// Mitsubishi GX Works2 project: MPS 장비 제어 4   PLC: Q03UDV

PROGRAM MAIN
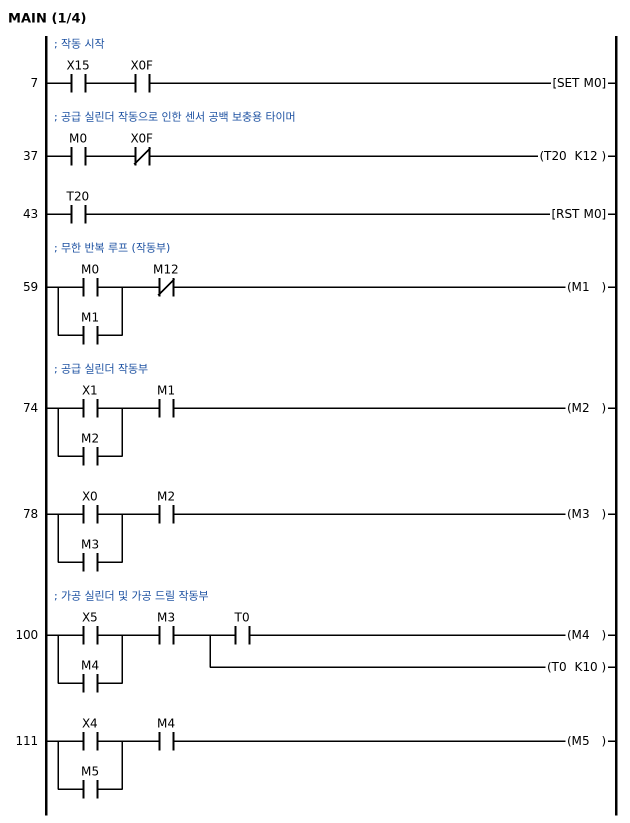
; 작동 시작
7     LD      X15
      AND     X0F
      SET     M0
; 공급 실린더 작동으로 인한 센서 공백 보충용 타이머
37    LD      M0
      ANI     X0F
      OUT     T20 K12
43    LD      T20
      RST     M0
; 무한 반복 루프 (작동부)
59    LD      M0
      OR      M1
      ANI     M12
      OUT     M1
; 공급 실린더 작동부
74    LD      X1
      OR      M2
      AND     M1
      OUT     M2
78    LD      X0
      OR      M3
      AND     M2
      OUT     M3
; 가공 실린더 및 가공 드릴 작동부
100   LD      X5
      OR      M4
      AND     M3
      MPS
      AND     T0
      OUT     M4
      MPP
      OUT     T0 K10
111   LD      X4
      OR      M5
      AND     M4
      OUT     M5
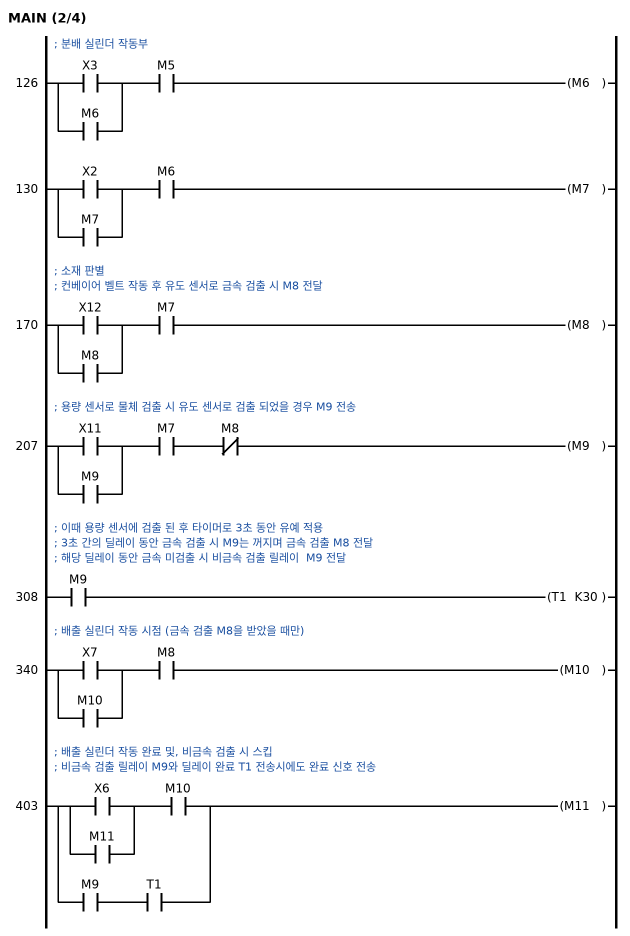
; 분배 실린더 작동부
126   LD      X3
      OR      M6
      AND     M5
      OUT     M6
130   LD      X2
      OR      M7
      AND     M6
      OUT     M7
; 소재 판별
; 컨베이어 벨트 작동 후 유도 센서로 금속 검출 시 M8 전달
170   LD      X12
      OR      M8
      AND     M7
      OUT     M8
; 용량 센서로 물체 검출 시 유도 센서로 검출 되었을 경우 M9 전송
207   LD      X11
      OR      M9
      AND     M7
      ANI     M8
      OUT     M9
; 이때 용량 센서에 검출 된 후 타이머로 3초 동안 유예 적용
; 3초 간의 딜레이 동안 금속 검출 시 M9는 꺼지며 금속 검출 M8 전달
; 해당 딜레이 동안 금속 미검출 시 비금속 검출 릴레이  M9 전달
308   LD      M9
      OUT     T1 K30
; 배출 실린더 작동 시점 (금속 검출 M8을 받았을 때만)
340   LD      X7
      OR      M10
      AND     M8
      OUT     M10
; 배출 실린더 작동 완료 및, 비금속 검출 시 스킵
; 비금속 검출 릴레이 M9와 딜레이 완료 T1 전송시에도 완료 신호 전송
403   LD      X6
      OR      M11
      AND     M10
      LD      M9
      AND     T1
      ORB
      OUT     M11
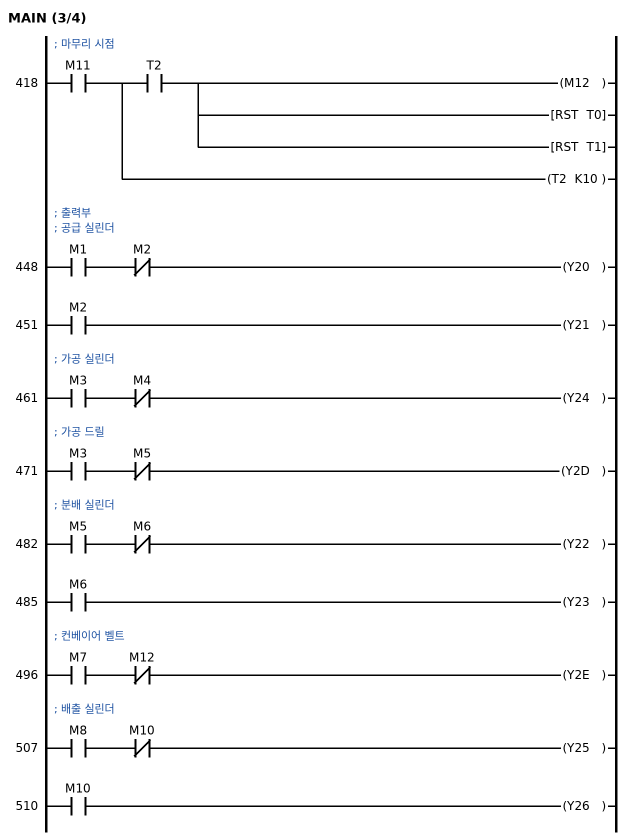
; 마무리 시점
418   LD      M11
      MPS
      AND     T2
      OUT     M12
      RST     T0
      RST     T1
      MPP
      OUT     T2 K10
; 출력부
; 공급 실린더
448   LD      M1
      ANI     M2
      OUT     Y20
451   LD      M2
      OUT     Y21
; 가공 실린더
461   LD      M3
      ANI     M4
      OUT     Y24
; 가공 드릴
471   LD      M3
      ANI     M5
      OUT     Y2D
; 분배 실린더
482   LD      M5
      ANI     M6
      OUT     Y22
485   LD      M6
      OUT     Y23
; 컨베이어 벨트
496   LD      M7
      ANI     M12
      OUT     Y2E
; 배출 실린더
507   LD      M8
      ANI     M10
      OUT     Y25
510   LD      M10
      OUT     Y26
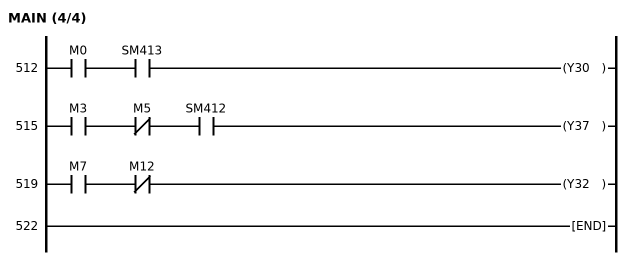
512   LD      M0
      AND     SM413
      OUT     Y30
515   LD      M3
      ANI     M5
      AND     SM412
      OUT     Y37
519   LD      M7
      ANI     M12
      OUT     Y32
522   END
END_PROGRAM
